PROGRAM POU_DALI_Prog
VAR
	fbDALI102Dimmer1Switch	 : FB_DALI102Dimmer1Switch(POU_Comm.fbKL6821Communication);
	bInitialize              : BOOL := FALSE;
	motionSensor			 : BOOL;
 	bRecallMaxLevel          : BOOL;
 	bRecallMinLevel          : BOOL;
 	//bOn                      : BOOL;
 	//bOff                     : BOOL;
  	bToggle                  : BOOL;
  	bGoToScene               : BOOL;
  	nScene                   : BYTE;
  	bSetLevel                : BOOL;
  	nLevel                   : BYTE := 254;
  	nLevelMemoryMode         : BYTE := 70;
  	nReferenceDeviceAddress  : BYTE;
  	tCycleActualLevel        : TIME := T#5S;
  	nOptions                 : DWORD := 0;
	nActualLevel             : BYTE;
END_VAR

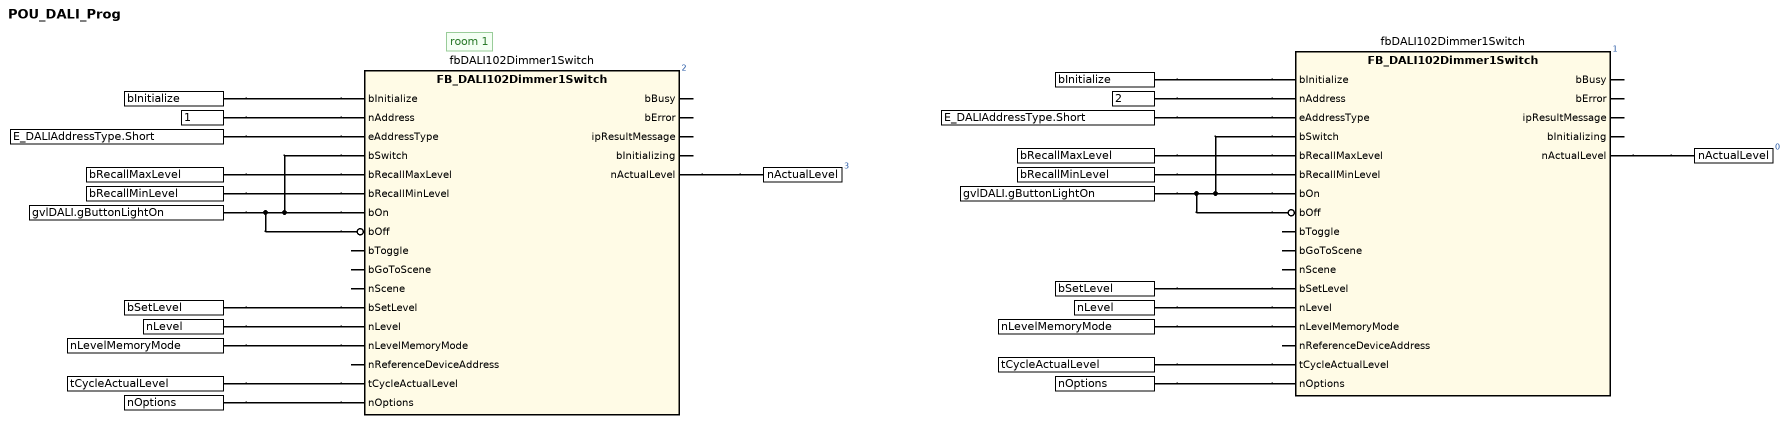
nActualLevel := fbDALI102Dimmer1Switch.nActualLevel;
fbDALI102Dimmer1Switch(
    bInitialize := bInitialize,
    nAddress := 2,
    eAddressType := E_DALIAddressType.Short,
    bSwitch := gvlDALI.gButtonLightOn,
    bRecallMaxLevel := bRecallMaxLevel,
    bRecallMinLevel := bRecallMinLevel,
    bOn := gvlDALI.gButtonLightOn,
    bOff := NOT gvlDALI.gButtonLightOn,
    bSetLevel := bSetLevel,
    nLevel := nLevel,
    nLevelMemoryMode := nLevelMemoryMode,
    tCycleActualLevel := tCycleActualLevel,
    nOptions := nOptions); // FB_DALI102Dimmer1Switch
// room 1
fbDALI102Dimmer1Switch(
    bInitialize := bInitialize,
    nAddress := 1,
    eAddressType := E_DALIAddressType.Short,
    bSwitch := gvlDALI.gButtonLightOn,
    bRecallMaxLevel := bRecallMaxLevel,
    bRecallMinLevel := bRecallMinLevel,
    bOn := gvlDALI.gButtonLightOn,
    bOff := NOT gvlDALI.gButtonLightOn,
    bSetLevel := bSetLevel,
    nLevel := nLevel,
    nLevelMemoryMode := nLevelMemoryMode,
    tCycleActualLevel := tCycleActualLevel,
    nOptions := nOptions); // FB_DALI102Dimmer1Switch
nActualLevel := fbDALI102Dimmer1Switch.nActualLevel;

END_PROGRAM

(* stored: Version 1.1.0.1, ProductVersion 3.1.4024.15
   POU POU_DALI_Prog: Id {4f67a694-1c35-4c24-9ca3-e16be0c42255}, SpecialFunc None *)
